SUBAPPLICATION Tuple (* Subapplication Type *)
  (* Standard: 61499-2 *)
  (* Version 1.0, 2023-02-17, Franz *)
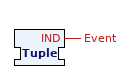
  EVENT_OUTPUT
    IND;
  END_EVENT
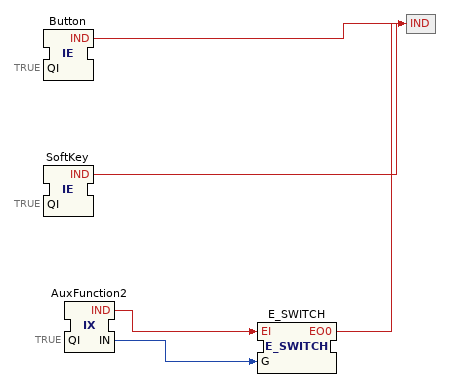
  FBS
    Button : eclipse4diac::io::IE(QI := TRUE);
    SoftKey : eclipse4diac::io::IE(QI := TRUE);
    AuxFunction2 : eclipse4diac::io::IX(QI := TRUE);
    E_SWITCH : iec61499::events::E_SWITCH;
  END_FBS
  EVENT_CONNECTIONS
    Button.IND TO IND;
    SoftKey.IND TO IND;
    AuxFunction2.IND TO E_SWITCH.EI;
    E_SWITCH.EO0 TO IND;
  END_CONNECTIONS
  DATA_CONNECTIONS
    AuxFunction2.IN TO E_SWITCH.G;
  END_CONNECTIONS
END_SUBAPPLICATION
